Staubli VAL3: Place.pgx

program place()
  local bool l_bNoError
  local joint l_jAppro
  local num l_nConvNum
  local num l_nError
  local num l_nMoveID
  local num l_nTrackStatus
  local pointRs l_pAppro
  local pointRs l_pPlace
  local string l_sToolStatus
begin
  l_nConvNum=1
  link(l_pPlace,world)
  //che modify start
  if nPlaceNum<0
    nPlaceNum=3
  endIf
  _mLoad=mLoad
  _mLoad.vel=mLoad.vel*nLoadRatio[nPlaceNum]
  _mLoad.accel=mLoad.accel*nLoadRatio[nPlaceNum]*nLoadRatio[nPlaceNum]
  _mLoad.decel=mLoad.decel*nLoadRatio[nPlaceNum]*nLoadRatio[nPlaceNum]

  //dControlVacuum[nPlaceNum]=false
  l_pPlace=pPlace[nPlaceNum]
  //end
  // Place part
  l_pAppro=appro(l_pPlace,{0,0,-nPlaceAppro,0,0,0})
  l_bNoError=pointToJoint(tGripper,jHome,l_pAppro,l_jAppro)
  call mot:getTrackStatus(l_nTrackStatus)
  if l_nTrackStatus>0
    // Use trackOff if the robot is synchronized
    if l_bNoError
      call mot:trackOffJ(l_jAppro,tGripper,_mLoad,l_nMoveID,l_nError)
    else
      call mot:trackOff(l_pAppro,tGripper,_mLoad,l_nMoveID,l_nError)
    endIf
  else
    // Use movej if the robot is not synchronized
    if l_bNoError
      l_nMoveID=movej(l_jAppro,tGripper,_mLoad)
    else
      l_nMoveID=movej(l_pAppro,tGripper,_mLoad)
    endIf
  endIf
  // wait permit signal
  //
  wait(dPermitPlace[nPlaceNum]==true)
  l_nMoveID=movel(l_pPlace,tGripper,mPlaceDown)
  wait(getMoveId()>l_nMoveID+nBlowID)
  _nBlowDelay=0.3
  waitEndMove()
  delay(nStopTime)
  l_nMoveID=movel(l_pAppro,tGripper,mPlaceUp)
  // check PartInTool if bPickDetection
  if bPickDetection
    //wait(getMoveId()>l_nMoveID-0.8)
    wait(getMoveId()>l_nMoveID+nBlowID-1.2)
    call getToolStatus(l_sToolStatus)
  else
    //wait(getMoveId()>l_nMoveID-0.2)
    wait(getMoveId()>l_nMoveID+nBlowID-1.2)
    _bPartInTool=false
  endIf
  // send done signal
  //dPlaceDone[nPlaceNum]=true
  wait(getMoveId()>l_nMoveID+0.1)
  delay(0)
  //dPlaceDone[nPlaceNum]=false
  if l_sToolStatus=="PartInTool" or _bPartInTool==false
    // A part has been placed
    _nCntPartsDone[l_nConvNum]=_nCntPartsDone[l_nConvNum]+1
  endIf
  delay(0)

  dPlaceDone[nPlaceNum]=true
  wait(getMoveId()>l_nMoveID+0.4)
  if nPlaceNum==3 and bSyn
    do
      sString=synServer
    until (sString=="done")
  endIf
  if nPlaceNum==0
    synServer="done"
  endIf
  nPlaceNum=nPlaceNum-1
  nTestData[4]=nTestData[4]+1
  //end

end
